PROGRAM MAIN
VAR
	cycleManager :CNM_CycleManager.SimpleCycleManager;
	interfaceTests :CNM_CycleManagerInterfacesTests.InterfaceTests(cycleManager);
END_VAR

TcUnit.RUN();

END_PROGRAM

(* stored: Version 1.1.0.1
   POU MAIN: Id {2c063c6d-39bb-4d22-8b03-82600500862b}, SpecialFunc None *)
